% RSLogix 500 project VeneerSander2017307.RSS, saved by version 8.30.00.16 %
PROJECT "UNTITLED"    % processor: Bul.1763 MicroLogix 1100 Series B %

PROGRAM FILES
  LAD 2 "MAIN"  8 rungs
  LAD 3 "OSC_SOL"  4 rungs
  LAD 4 "PRE1"  2 rungs
  LAD 5 "PRE2"  2 rungs
  LAD 6 "PRE3"  2 rungs
  LAD 9 "HMI"  11 rungs  % InputOutput States and other ifo %
  LAD 10 "VFD1"  7 rungs
  LAD 11 "VFD2"  7 rungs
  LAD 12 "Z_AXIS"  11 rungs

DATA FILES
  O0 OUTPUT  5 elements
  I1 INPUT  6 elements
  S2 STATUS  66 elements
  B3 BINARY  15 elements
  T4 TIMER  1 elements
  C5 COUNTER  1 elements
  R6 CONTROL  1 elements
  N7 INTEGER  1 elements
  F8 FLOAT  1 elements

LADDER 2 "MAIN"
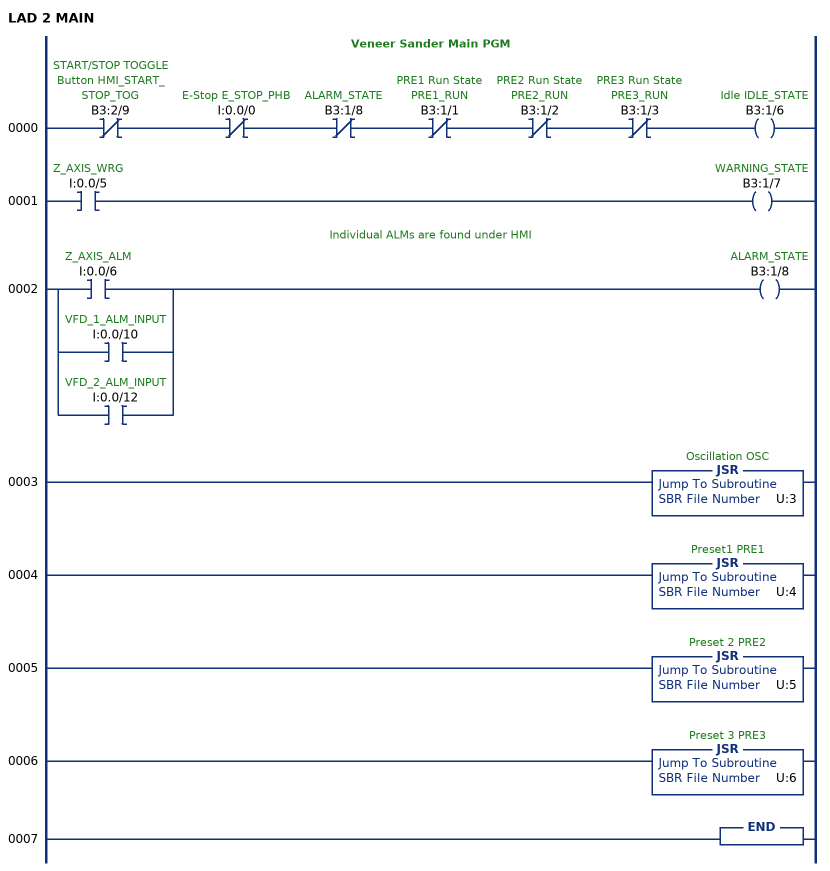
% Rung: 0 %  % edit flag set %
% TITLE: Veneer Sander Main PGM %
SOR XIO B3:2/9 XIO I:0.0/0 XIO B3:1/8 XIO B3:1/1 XIO B3:1/2 XIO B3:1/3 OTE B3:1/6 EOR
%   B3:2/9  HMI_START_STOP_TOG  "START/STOP TOGGLE Button" %
%   I:0.0/0  E_STOP_PHB  "E-Stop" %
%   B3:1/8  ALARM_STATE %
%   B3:1/1  PRE1_RUN  "PRE1 Run State" %
%   B3:1/2  PRE2_RUN  "PRE2 Run State" %
%   B3:1/3  PRE3_RUN  "PRE3 Run State" %
%   B3:1/6  IDLE_STATE  "Idle" %
% Rung: 1 %
SOR XIC I:0.0/5 OTE B3:1/7 EOR
%   I:0.0/5  Z_AXIS_WRG %
%   B3:1/7  WARNING_STATE %
% Rung: 2 %
% Individual ALMs are found under HMI %
SOR BST XIC I:0.0/6 NXB XIC I:0.0/10 NXB XIC I:0.0/12 BND OTE B3:1/8 EOR
%   I:0.0/6  Z_AXIS_ALM %
%   I:0.0/10  VFD_1_ALM_INPUT %
%   I:0.0/12  VFD_2_ALM_INPUT %
%   B3:1/8  ALARM_STATE %
% Rung: 3 %
SOR JSR U:3 EOR
%   U:3  OSC  "Oscillation" %
% Rung: 4 %
SOR JSR U:4 EOR
%   U:4  PRE1  "Preset1" %
% Rung: 5 %
SOR JSR U:5 EOR
%   U:5  PRE2  "Preset 2" %
% Rung: 6 %
SOR JSR U:6 EOR
%   U:6  PRE3  "Preset 3" %
% Rung: 7 %
SOR END EOR

LADDER 3 "OSC_SOL"
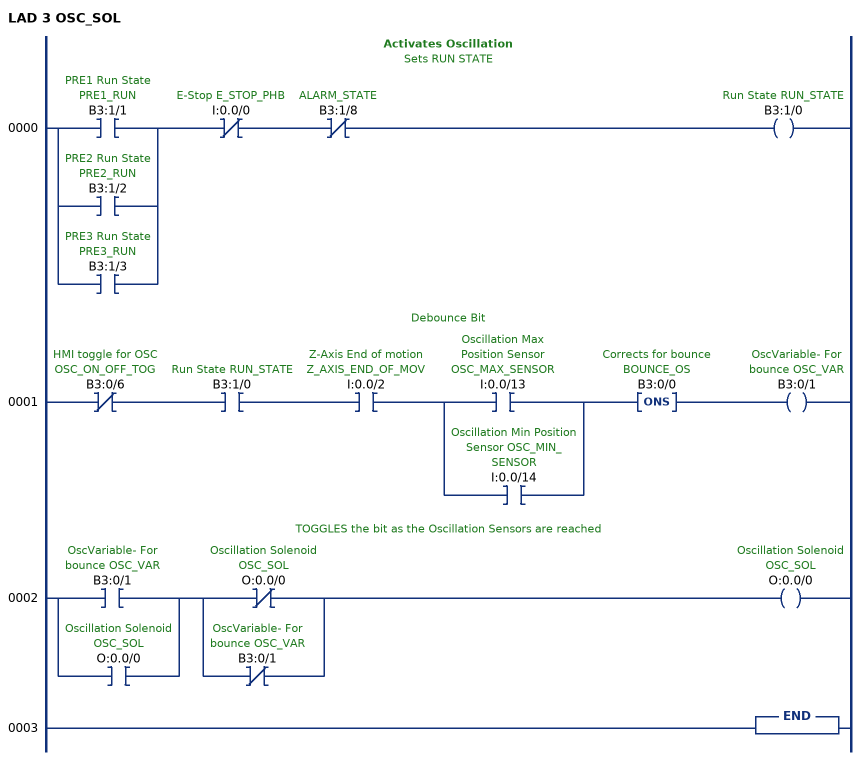
% Rung: 0 %  % edit flag set %
% TITLE: Activates Oscillation %
% Sets RUN STATE %
SOR BST XIC B3:1/1 NXB XIC B3:1/2 NXB XIC B3:1/3 BND XIO I:0.0/0 XIO B3:1/8 OTE B3:1/0 EOR
%   B3:1/1  PRE1_RUN  "PRE1 Run State" %
%   B3:1/2  PRE2_RUN  "PRE2 Run State" %
%   B3:1/3  PRE3_RUN  "PRE3 Run State" %
%   I:0.0/0  E_STOP_PHB  "E-Stop" %
%   B3:1/8  ALARM_STATE %
%   B3:1/0  RUN_STATE  "Run State" %
% Rung: 1 %  % edit flag set %
% Debounce Bit %
SOR XIO B3:0/6 XIC B3:1/0 XIC I:0.0/2 BST XIC I:0.0/13 NXB XIC I:0.0/14 BND ONS B3:0/0 OTE B3:0/1 EOR
%   B3:0/6  OSC_ON_OFF_TOG  "HMI toggle for OSC" %
%   B3:1/0  RUN_STATE  "Run State" %
%   I:0.0/2  Z_AXIS_END_OF_MOV  "Z-Axis End of motion" %
%   I:0.0/13  OSC_MAX_SENSOR  "Oscillation Max Position Sensor" %
%   I:0.0/14  OSC_MIN_SENSOR  "Oscillation Min Position Sensor" %
%   B3:0/0  BOUNCE_OS  "Corrects for bounce" %
%   B3:0/1  OSC_VAR  "OscVariable- For bounce" %
% Rung: 2 %
% TOGGLES the bit as the Oscillation Sensors are reached %
SOR BST XIC B3:0/1 NXB XIC O:0.0/0 BND BST XIO O:0.0/0 NXB XIO B3:0/1 BND OTE O:0.0/0 EOR
%   B3:0/1  OSC_VAR  "OscVariable- For bounce" %
%   O:0.0/0  OSC_SOL  "Oscillation Solenoid" %
% Rung: 3 %
SOR END EOR

LADDER 4 "PRE1"
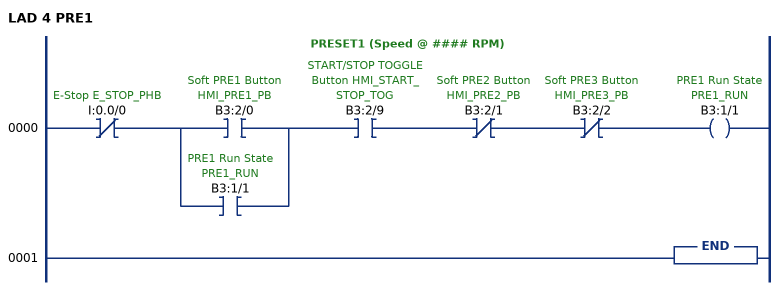
% Rung: 0 %  % edit flag set %
% TITLE: PRESET1 (Speed @ #### RPM) %
SOR XIO I:0.0/0 BST XIC B3:2/0 NXB XIC B3:1/1 BND XIC B3:2/9 XIO B3:2/1 XIO B3:2/2 OTE B3:1/1 EOR
%   I:0.0/0  E_STOP_PHB  "E-Stop" %
%   B3:2/0  HMI_PRE1_PB  "Soft PRE1 Button" %
%   B3:1/1  PRE1_RUN  "PRE1 Run State" %
%   B3:2/9  HMI_START_STOP_TOG  "START/STOP TOGGLE Button" %
%   B3:2/1  HMI_PRE2_PB  "Soft PRE2 Button" %
%   B3:2/2  HMI_PRE3_PB  "Soft PRE3 Button" %
% Rung: 1 %
SOR END EOR

LADDER 5 "PRE2"
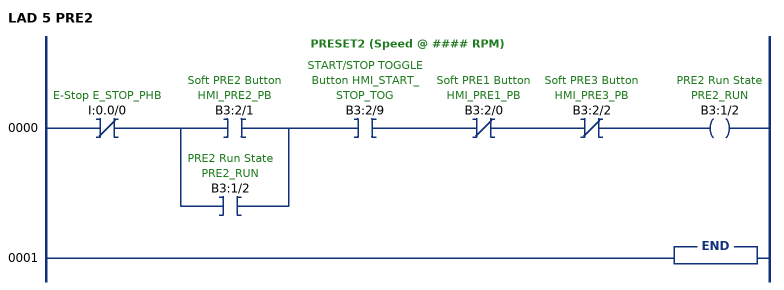
% Rung: 0 %  % edit flag set %
% TITLE: PRESET2 (Speed @ #### RPM) %
SOR XIO I:0.0/0 BST XIC B3:2/1 NXB XIC B3:1/2 BND XIC B3:2/9 XIO B3:2/0 XIO B3:2/2 OTE B3:1/2 EOR
%   I:0.0/0  E_STOP_PHB  "E-Stop" %
%   B3:2/1  HMI_PRE2_PB  "Soft PRE2 Button" %
%   B3:1/2  PRE2_RUN  "PRE2 Run State" %
%   B3:2/9  HMI_START_STOP_TOG  "START/STOP TOGGLE Button" %
%   B3:2/0  HMI_PRE1_PB  "Soft PRE1 Button" %
%   B3:2/2  HMI_PRE3_PB  "Soft PRE3 Button" %
% Rung: 1 %
SOR END EOR

LADDER 6 "PRE3"
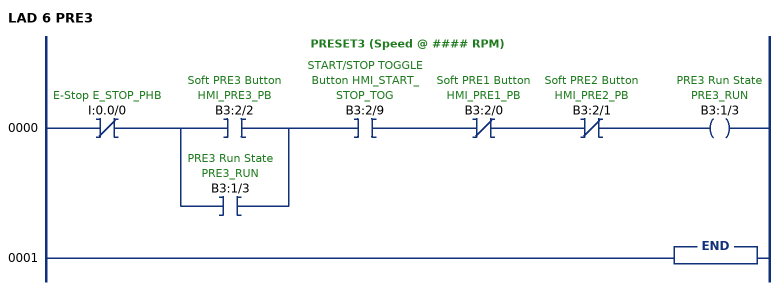
% Rung: 0 %  % edit flag set %
% TITLE: PRESET3 (Speed @ #### RPM) %
SOR XIO I:0.0/0 BST XIC B3:2/2 NXB XIC B3:1/3 BND XIC B3:2/9 XIO B3:2/0 XIO B3:2/1 OTE B3:1/3 EOR
%   I:0.0/0  E_STOP_PHB  "E-Stop" %
%   B3:2/2  HMI_PRE3_PB  "Soft PRE3 Button" %
%   B3:1/3  PRE3_RUN  "PRE3 Run State" %
%   B3:2/9  HMI_START_STOP_TOG  "START/STOP TOGGLE Button" %
%   B3:2/0  HMI_PRE1_PB  "Soft PRE1 Button" %
%   B3:2/1  HMI_PRE2_PB  "Soft PRE2 Button" %
% Rung: 1 %
SOR END EOR

LADDER 9 "HMI"    % InputOutput States and other ifo %
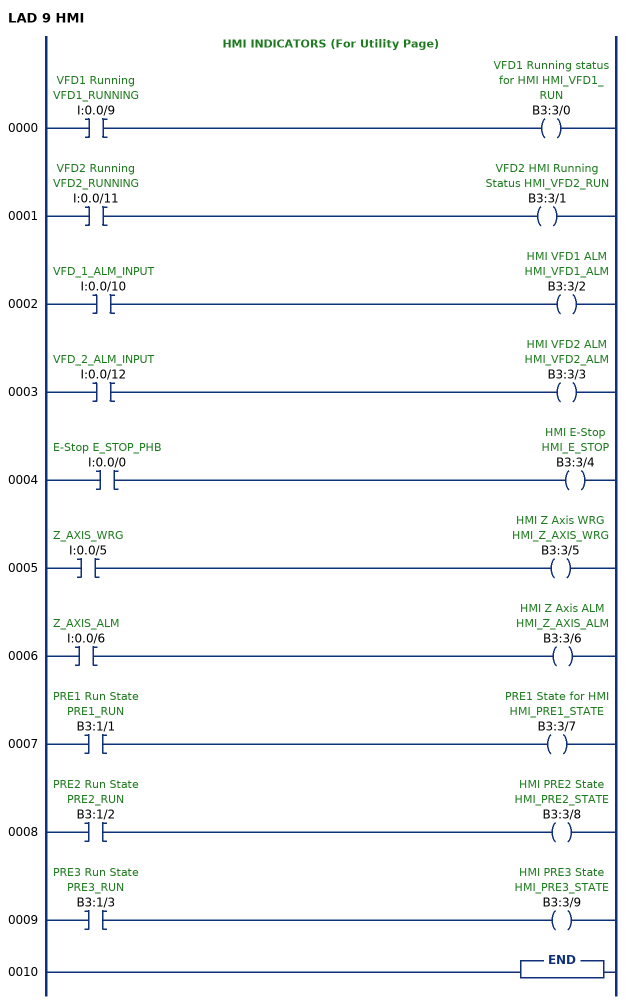
% Rung: 0 %
% TITLE: HMI INDICATORS (For Utility Page) %
SOR XIC I:0.0/9 OTE B3:3/0 EOR
%   I:0.0/9  VFD1_RUNNING  "VFD1 Running" %
%   B3:3/0  HMI_VFD1_RUN  "VFD1 Running status for HMI" %
% Rung: 1 %
SOR XIC I:0.0/11 OTE B3:3/1 EOR
%   I:0.0/11  VFD2_RUNNING  "VFD2 Running" %
%   B3:3/1  HMI_VFD2_RUN  "VFD2 HMI Running Status" %
% Rung: 2 %
SOR XIC I:0.0/10 OTE B3:3/2 EOR
%   I:0.0/10  VFD_1_ALM_INPUT %
%   B3:3/2  HMI_VFD1_ALM  "HMI VFD1 ALM" %
% Rung: 3 %
SOR XIC I:0.0/12 OTE B3:3/3 EOR
%   I:0.0/12  VFD_2_ALM_INPUT %
%   B3:3/3  HMI_VFD2_ALM  "HMI VFD2 ALM" %
% Rung: 4 %
SOR XIC I:0.0/0 OTE B3:3/4 EOR
%   I:0.0/0  E_STOP_PHB  "E-Stop" %
%   B3:3/4  HMI_E_STOP  "HMI E-Stop" %
% Rung: 5 %
SOR XIC I:0.0/5 OTE B3:3/5 EOR
%   I:0.0/5  Z_AXIS_WRG %
%   B3:3/5  HMI_Z_AXIS_WRG  "HMI Z Axis WRG" %
% Rung: 6 %
SOR XIC I:0.0/6 OTE B3:3/6 EOR
%   I:0.0/6  Z_AXIS_ALM %
%   B3:3/6  HMI_Z_AXIS_ALM  "HMI Z Axis ALM" %
% Rung: 7 %
SOR XIC B3:1/1 OTE B3:3/7 EOR
%   B3:1/1  PRE1_RUN  "PRE1 Run State" %
%   B3:3/7  HMI_PRE1_STATE  "PRE1 State for HMI" %
% Rung: 8 %
SOR XIC B3:1/2 OTE B3:3/8 EOR
%   B3:1/2  PRE2_RUN  "PRE2 Run State" %
%   B3:3/8  HMI_PRE2_STATE  "HMI PRE2 State" %
% Rung: 9 %
SOR XIC B3:1/3 OTE B3:3/9 EOR
%   B3:1/3  PRE3_RUN  "PRE3 Run State" %
%   B3:3/9  HMI_PRE3_STATE  "HMI PRE3 State" %
% Rung: 10 %
SOR END EOR

LADDER 10 "VFD1"
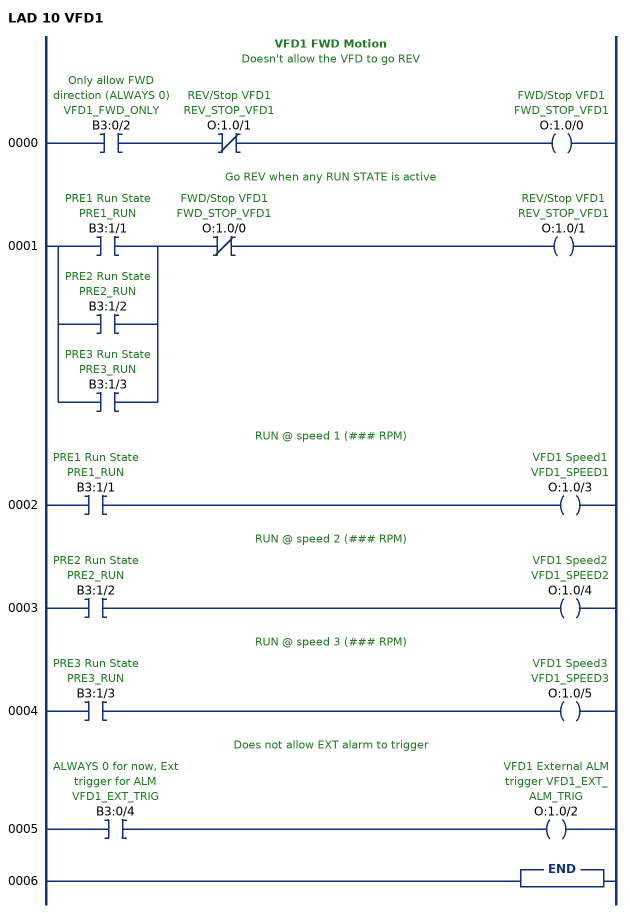
% Rung: 0 %
% TITLE: VFD1 FWD Motion %
% Doesn't allow the VFD to go REV %
SOR XIC B3:0/2 XIO O:1.0/1 OTE O:1.0/0 EOR
%   B3:0/2  VFD1_FWD_ONLY  "Only allow FWD direction (ALWAYS 0)" %
%   O:1.0/1  REV_STOP_VFD1  "REV/Stop VFD1" %
%   O:1.0/0  FWD_STOP_VFD1  "FWD/Stop VFD1" %
% Rung: 1 %
% Go REV when any RUN STATE is active %
SOR BST XIC B3:1/1 NXB XIC B3:1/2 NXB XIC B3:1/3 BND XIO O:1.0/0 OTE O:1.0/1 EOR
%   B3:1/1  PRE1_RUN  "PRE1 Run State" %
%   B3:1/2  PRE2_RUN  "PRE2 Run State" %
%   B3:1/3  PRE3_RUN  "PRE3 Run State" %
%   O:1.0/0  FWD_STOP_VFD1  "FWD/Stop VFD1" %
%   O:1.0/1  REV_STOP_VFD1  "REV/Stop VFD1" %
% Rung: 2 %
% RUN @ speed 1 (### RPM) %
SOR XIC B3:1/1 OTE O:1.0/3 EOR
%   B3:1/1  PRE1_RUN  "PRE1 Run State" %
%   O:1.0/3  VFD1_SPEED1  "VFD1 Speed1" %
% Rung: 3 %
% RUN @ speed 2 (### RPM) %
SOR XIC B3:1/2 OTE O:1.0/4 EOR
%   B3:1/2  PRE2_RUN  "PRE2 Run State" %
%   O:1.0/4  VFD1_SPEED2  "VFD1 Speed2" %
% Rung: 4 %
% RUN @ speed 3 (### RPM) %
SOR XIC B3:1/3 OTE O:1.0/5 EOR
%   B3:1/3  PRE3_RUN  "PRE3 Run State" %
%   O:1.0/5  VFD1_SPEED3  "VFD1 Speed3" %
% Rung: 5 %
% Does not allow EXT alarm to trigger %
SOR XIC B3:0/4 OTE O:1.0/2 EOR
%   B3:0/4  VFD1_EXT_TRIG  "ALWAYS 0 for now, Ext trigger for ALM" %
%   O:1.0/2  VFD1_EXT_ALM_TRIG  "VFD1 External ALM trigger" %
% Rung: 6 %
SOR END EOR

LADDER 11 "VFD2"
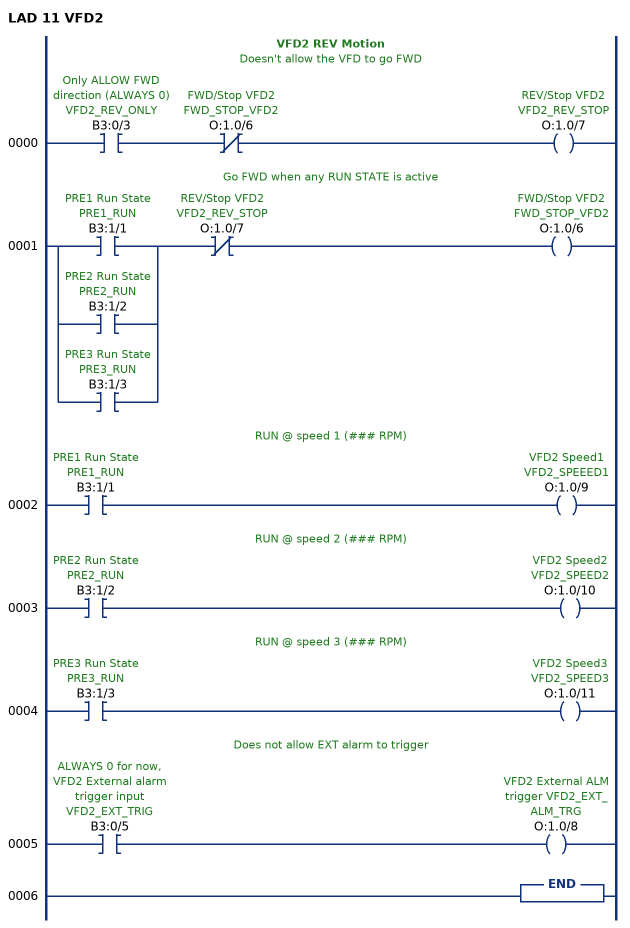
% Rung: 0 %
% TITLE: VFD2 REV Motion %
% Doesn't allow the VFD to go FWD %
SOR XIC B3:0/3 XIO O:1.0/6 OTE O:1.0/7 EOR
%   B3:0/3  VFD2_REV_ONLY  "Only ALLOW FWD direction (ALWAYS 0)" %
%   O:1.0/6  FWD_STOP_VFD2  "FWD/Stop VFD2" %
%   O:1.0/7  VFD2_REV_STOP  "REV/Stop VFD2" %
% Rung: 1 %
% Go FWD when any RUN STATE is active %
SOR BST XIC B3:1/1 NXB XIC B3:1/2 NXB XIC B3:1/3 BND XIO O:1.0/7 OTE O:1.0/6 EOR
%   B3:1/1  PRE1_RUN  "PRE1 Run State" %
%   B3:1/2  PRE2_RUN  "PRE2 Run State" %
%   B3:1/3  PRE3_RUN  "PRE3 Run State" %
%   O:1.0/7  VFD2_REV_STOP  "REV/Stop VFD2" %
%   O:1.0/6  FWD_STOP_VFD2  "FWD/Stop VFD2" %
% Rung: 2 %
% RUN @ speed 1 (### RPM) %
SOR XIC B3:1/1 OTE O:1.0/9 EOR
%   B3:1/1  PRE1_RUN  "PRE1 Run State" %
%   O:1.0/9  VFD2_SPEEED1  "VFD2 Speed1" %
% Rung: 3 %
% RUN @ speed 2 (### RPM) %
SOR XIC B3:1/2 OTE O:1.0/10 EOR
%   B3:1/2  PRE2_RUN  "PRE2 Run State" %
%   O:1.0/10  VFD2_SPEED2  "VFD2 Speed2" %
% Rung: 4 %
% RUN @ speed 3 (### RPM) %
SOR XIC B3:1/3 OTE O:1.0/11 EOR
%   B3:1/3  PRE3_RUN  "PRE3 Run State" %
%   O:1.0/11  VFD2_SPEED3  "VFD2 Speed3" %
% Rung: 5 %
% Does not allow EXT alarm to trigger %
SOR XIC B3:0/5 OTE O:1.0/8 EOR
%   B3:0/5  VFD2_EXT_TRIG  "ALWAYS 0 for now, VFD2 External alarm trigger input" %
%   O:1.0/8  VFD2_EXT_ALM_TRG  "VFD2 External ALM trigger" %
% Rung: 6 %
SOR END EOR

LADDER 12 "Z_AXIS"
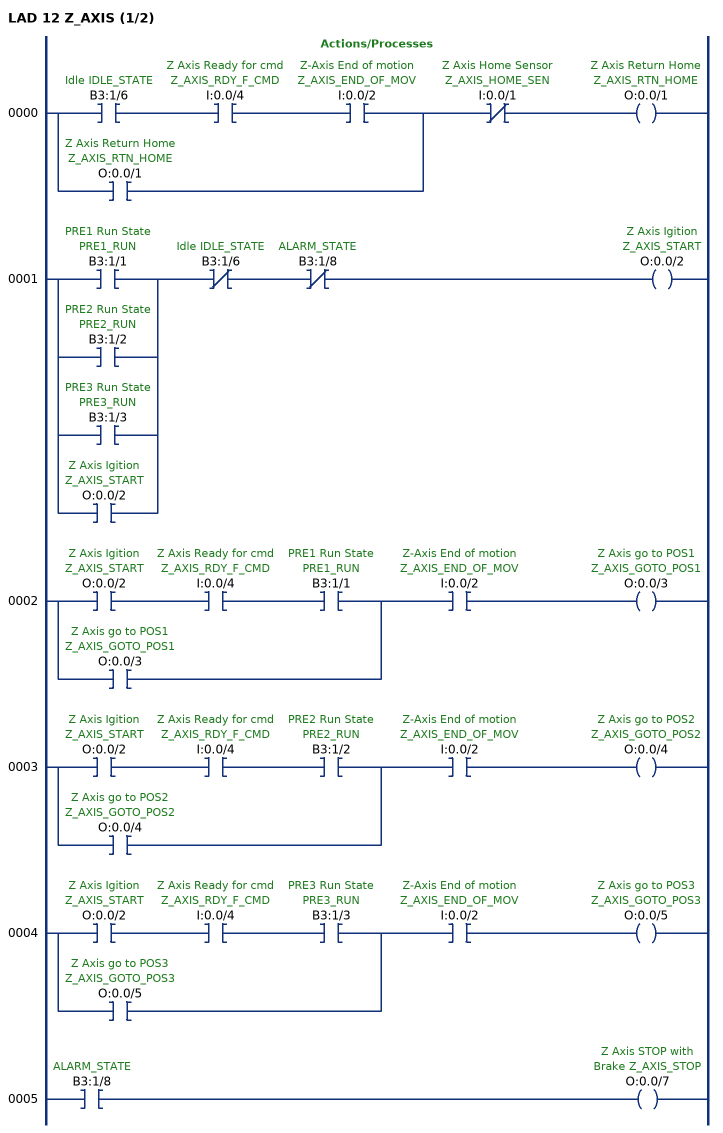
% Rung: 0 %
% TITLE: Actions/Processes %
SOR BST XIC B3:1/6 XIC I:0.0/4 XIC I:0.0/2 NXB XIC O:0.0/1 BND XIO I:0.0/1 OTE O:0.0/1 EOR
%   B3:1/6  IDLE_STATE  "Idle" %
%   I:0.0/4  Z_AXIS_RDY_F_CMD  "Z Axis Ready for cmd" %
%   I:0.0/2  Z_AXIS_END_OF_MOV  "Z-Axis End of motion" %
%   O:0.0/1  Z_AXIS_RTN_HOME  "Z Axis Return Home" %
%   I:0.0/1  Z_AXIS_HOME_SEN  "Z Axis Home Sensor" %
% Rung: 1 %
SOR BST XIC B3:1/1 NXB XIC B3:1/2 NXB XIC B3:1/3 NXB XIC O:0.0/2 BND XIO B3:1/6 XIO B3:1/8 OTE O:0.0/2 EOR
%   B3:1/1  PRE1_RUN  "PRE1 Run State" %
%   B3:1/2  PRE2_RUN  "PRE2 Run State" %
%   B3:1/3  PRE3_RUN  "PRE3 Run State" %
%   O:0.0/2  Z_AXIS_START  "Z Axis Igition" %
%   B3:1/6  IDLE_STATE  "Idle" %
%   B3:1/8  ALARM_STATE %
% Rung: 2 %
SOR BST XIC O:0.0/2 XIC I:0.0/4 XIC B3:1/1 NXB XIC O:0.0/3 BND XIC I:0.0/2 OTE O:0.0/3 EOR
%   O:0.0/2  Z_AXIS_START  "Z Axis Igition" %
%   I:0.0/4  Z_AXIS_RDY_F_CMD  "Z Axis Ready for cmd" %
%   B3:1/1  PRE1_RUN  "PRE1 Run State" %
%   O:0.0/3  Z_AXIS_GOTO_POS1  "Z Axis go to POS1" %
%   I:0.0/2  Z_AXIS_END_OF_MOV  "Z-Axis End of motion" %
% Rung: 3 %  % edit flag set %
SOR BST XIC O:0.0/2 XIC I:0.0/4 XIC B3:1/2 NXB XIC O:0.0/4 BND XIC I:0.0/2 OTE O:0.0/4 EOR
%   O:0.0/2  Z_AXIS_START  "Z Axis Igition" %
%   I:0.0/4  Z_AXIS_RDY_F_CMD  "Z Axis Ready for cmd" %
%   B3:1/2  PRE2_RUN  "PRE2 Run State" %
%   O:0.0/4  Z_AXIS_GOTO_POS2  "Z Axis go to POS2" %
%   I:0.0/2  Z_AXIS_END_OF_MOV  "Z-Axis End of motion" %
% Rung: 4 %  % edit flag set %
SOR BST XIC O:0.0/2 XIC I:0.0/4 XIC B3:1/3 NXB XIC O:0.0/5 BND XIC I:0.0/2 OTE O:0.0/5 EOR
%   O:0.0/2  Z_AXIS_START  "Z Axis Igition" %
%   I:0.0/4  Z_AXIS_RDY_F_CMD  "Z Axis Ready for cmd" %
%   B3:1/3  PRE3_RUN  "PRE3 Run State" %
%   O:0.0/5  Z_AXIS_GOTO_POS3  "Z Axis go to POS3" %
%   I:0.0/2  Z_AXIS_END_OF_MOV  "Z-Axis End of motion" %
% Rung: 5 %
SOR XIC B3:1/8 OTE O:0.0/7 EOR
%   B3:1/8  ALARM_STATE %
%   O:0.0/7  Z_AXIS_STOP  "Z Axis STOP with Brake" %

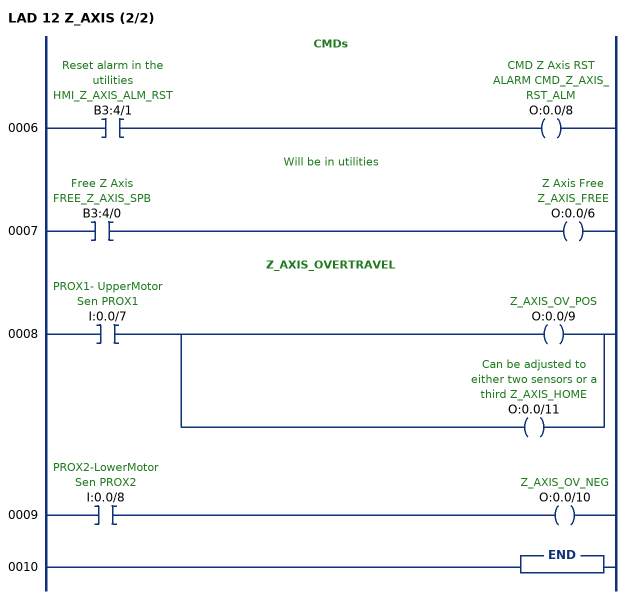
% Rung: 6 %
% TITLE: CMDs %
SOR XIC B3:4/1 OTE O:0.0/8 EOR
%   B3:4/1  HMI_Z_AXIS_ALM_RST  "Reset alarm in the utilities" %
%   O:0.0/8  CMD_Z_AXIS_RST_ALM  "CMD Z Axis RST ALARM" %
% Rung: 7 %
% Will be in utilities %
SOR XIC B3:4/0 OTE O:0.0/6 EOR
%   B3:4/0  FREE_Z_AXIS_SPB  "Free Z Axis" %
%   O:0.0/6  Z_AXIS_FREE  "Z Axis Free" %
% Rung: 8 %
% TITLE: Z_AXIS_OVERTRAVEL %
SOR XIC I:0.0/7 BST OTE O:0.0/9 NXB OTE O:0.0/11 BND EOR
%   I:0.0/7  PROX1  "PROX1- UpperMotorSen" %
%   O:0.0/9  Z_AXIS_OV_POS %
%   O:0.0/11  Z_AXIS_HOME  "Can be adjusted to either two sensors or a third" %
% Rung: 9 %
SOR XIC I:0.0/8 OTE O:0.0/10 EOR
%   I:0.0/8  PROX2  "PROX2-LowerMotorSen" %
%   O:0.0/10  Z_AXIS_OV_NEG %
% Rung: 10 %
SOR END EOR

OTHER DOCUMENTED ADDRESSES
  DFILE:0  "OUTPUT"
  DFILE:1  "INPUT"
  DFILE:2  "STATUS"
  DFILE:3  "BINARY"
  DFILE:4  "TIMER"
  DFILE:5  "COUNTER"
  DFILE:6  "CONTROL"
  DFILE:7  "INTEGER"
  DFILE:8  "FLOAT"
  I:0.0/3  Z_AXIS_IN_AREA1  "Z Axis in area 1"
  O:8  VFD2_ALARM  "VFD2 ALM"
  U:7  PRE4
  U:8  PRE5

REVISION NOTES
  0: First save, programmed OscSol
  1: Added PRESETS
  2: Saving for a restart- loaded HMI software, and for lunch
  3: Leaving the day (7/13/17)
  4: All Outputs are in place, Refined and organized Prog Files
  5: Done for the week, very close to the finish.
     
     VFD2 and Z axis, and refining
  6: Finishing up logic- Remove PRE4 and 5,Competed all logic,  Add comments, polishing
  7: Removed Stop Binary bit and Implemented START as a START/STOP TOGGLE switch, OSC ON/OFF TOGGLE, Made sure Idle State (now Return Home CMD) makes the Z axis go to HOME Position, Adjusted Descriptions, Reviewed for any errors and loops
